SUBAPPLICATION Uebung_012k_AIS (* String Input und Speichern INI mit Subapp (AIS Adapter) *)
  (* Standard: 61499-2; Description: Copyright (c) 2026 Meisterschulen am Ostbahnhof This program and the accompanying materials are made available under the terms of the Eclipse Public License 2.0 which is available at https://www.eclipse.org/legal/epl-2.0/ SPDX-License-Identifier: EPL-2.0 *)
  (* Version 1.0, 2026-04-24, Franz Höpfinger, Meisterschulen am Ostbahnhof, AIS adapter variant of Uebung_012k *)
  PACKAGE Uebungen;
  IMPORT Uebungen::const::NVS::NVS_Keys::KEY_I1_STORE;
  IMPORT Uebungen::const::NVS::NVS_Keys::SECTION_I1_STORE;
  IMPORT Uebungen::const::UT::DefaultPool::InputString_S1;
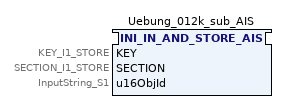
  SUBAPPS
    Uebung_012k_sub_AIS : MyLib::sys::INI_IN_AND_STORE_AIS(KEY := KEY_I1_STORE, SECTION := SECTION_I1_STORE, u16ObjId := InputString_S1);
  END_SUBAPPS
END_SUBAPPLICATION
